FUNCTION_BLOCK WKPC_GEN (* Random Workpiece Generator *)
  (* Standard: 61499-1; Classification: Simulation *)
  (* Version 0.2, 2004-09-16, JHC, Rockwell Automation, Generalized from PR_GEN. *)
  (* Version 0.1, 2004-08-06, JHC, Rockwell Automation, Changed PPEG to UINT. *)
  (* Version 0.0, 2002-04-11, JHC, Rockwell Automation *)
  (* Compiler header: package fb.rt.mva; *)
  (* Compiler Java Sun JDK 1.4.2 *)
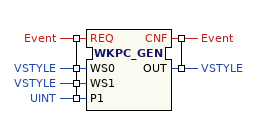
  EVENT_INPUT
    REQ WITH WS0, WS1, P1; (* Normal Execution Request *)
  END_EVENT
  EVENT_OUTPUT
    CNF WITH OUT; (* Execution Confirmation *)
  END_EVENT
  VAR_INPUT
    WS0 : VSTYLE := PEG; (* Workpiece Style 0 *)
    WS1 : VSTYLE := RING; (* Workpiece Style 1 *)
    P1 : UINT := 50; (* Probability that OUT=WS1 (0-100%) *)
  END_VAR
  VAR_OUTPUT
    OUT : VSTYLE := PEG;
  END_VAR
  ALGORITHM REQ IN Java:
OUT.value = ((Math.random()*100)<=P1.value)? WS1.value : WS0.value;
CNF.serviceEvent(this);
  END_ALGORITHM
END_FUNCTION_BLOCK
